SYSTEM OPCUAClient
  (* Version 1.0, Author, Eclipse 4diac *)
  APPLICATION OPCUAClientApp
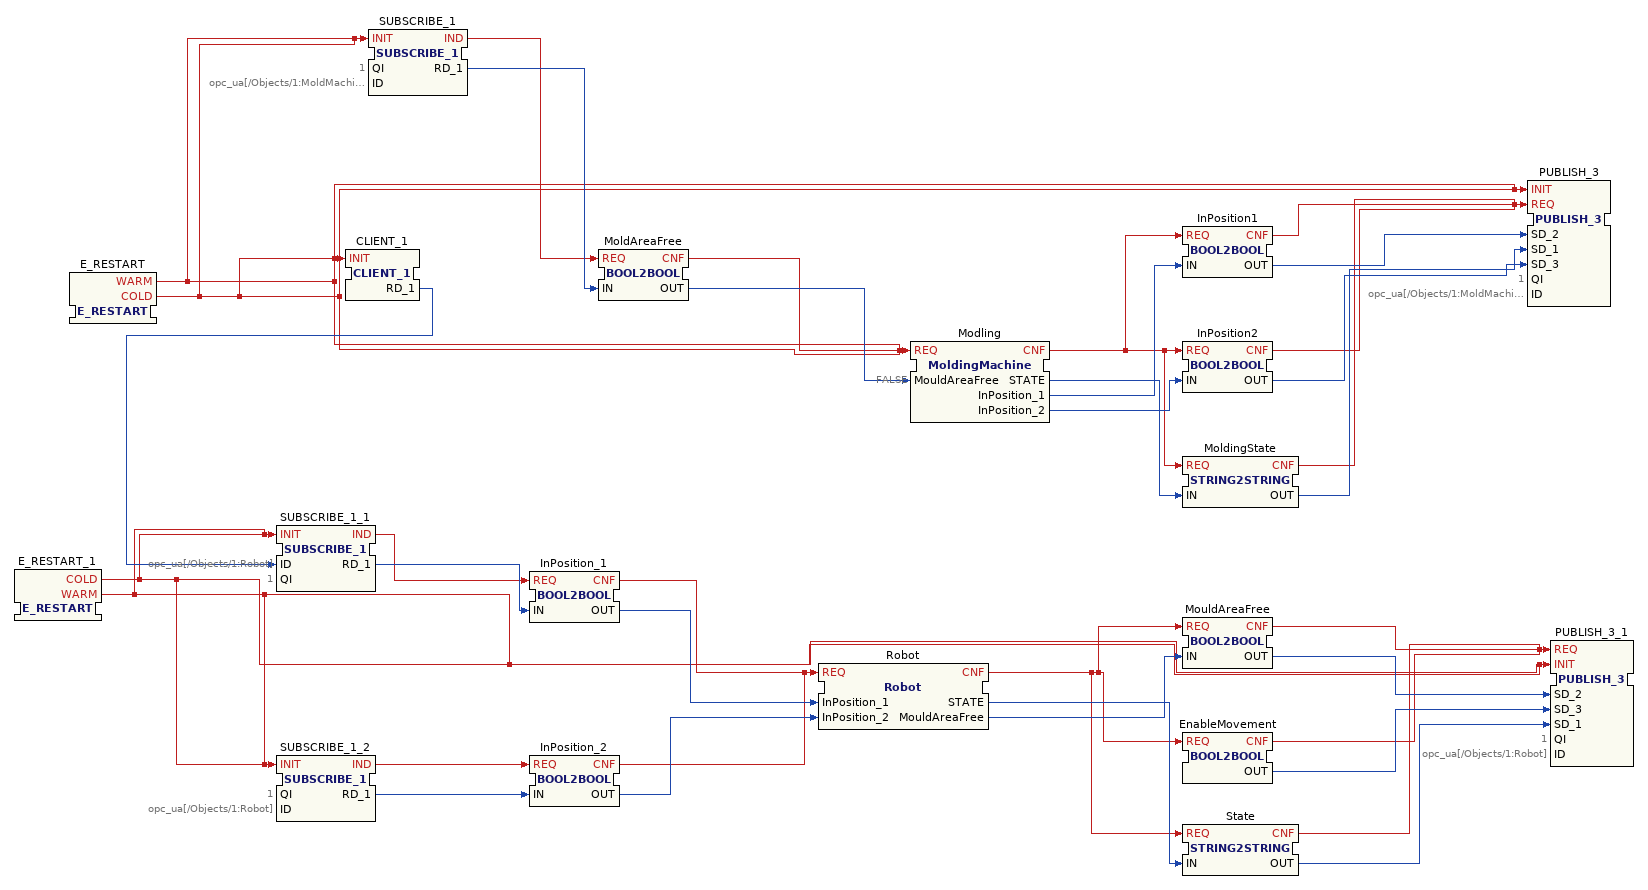
    FBS
      MoldAreaFree : BOOL2BOOL;
      E_RESTART : E_RESTART;
      SUBSCRIBE_1 : SUBSCRIBE_1(QI := 1, ID := opc_ua[/Objects/1:MoldMachine]);
      SUBSCRIBE_1_1 : SUBSCRIBE_1(QI := 1, ID := opc_ua[/Objects/1:Robot]);
      PUBLISH_3 : PUBLISH_3(QI := 1, ID := opc_ua[/Objects/1:MoldMachine]);
      Modling : MoldingMachine(MouldAreaFree := FALSE);
      InPosition_1 : BOOL2BOOL;
      SUBSCRIBE_1_2 : SUBSCRIBE_1(QI := 1, ID := opc_ua[/Objects/1:Robot]);
      InPosition_2 : BOOL2BOOL;
      PUBLISH_3_1 : PUBLISH_3(QI := 1, ID := opc_ua[/Objects/1:Robot]);
      InPosition1 : BOOL2BOOL;
      InPosition2 : BOOL2BOOL;
      MoldingState : STRING2STRING;
      MouldAreaFree : BOOL2BOOL;
      EnableMovement : BOOL2BOOL;
      State : STRING2STRING;
      Robot : Robot;
      E_RESTART_1 : E_RESTART;
      CLIENT_1 : CLIENT_1;
    END_FBS
    EVENT_CONNECTIONS
      E_RESTART.WARM TO SUBSCRIBE_1.INIT;
      E_RESTART.COLD TO SUBSCRIBE_1.INIT;
      SUBSCRIBE_1.IND TO MoldAreaFree.REQ;
      E_RESTART.COLD TO PUBLISH_3.INIT;
      E_RESTART.WARM TO PUBLISH_3.INIT;
      MoldAreaFree.CNF TO Modling.REQ;
      E_RESTART.COLD TO Modling.REQ;
      E_RESTART.WARM TO Modling.REQ;
      SUBSCRIBE_1_1.IND TO InPosition_1.REQ;
      SUBSCRIBE_1_2.IND TO InPosition_2.REQ;
      Modling.CNF TO InPosition1.REQ;
      Modling.CNF TO InPosition2.REQ;
      Modling.CNF TO MoldingState.REQ;
      InPosition1.CNF TO PUBLISH_3.REQ;
      InPosition2.CNF TO PUBLISH_3.REQ;
      MoldingState.CNF TO PUBLISH_3.REQ;
      InPosition_1.CNF TO Robot.REQ;
      InPosition_2.CNF TO Robot.REQ;
      Robot.CNF TO MouldAreaFree.REQ;
      Robot.CNF TO EnableMovement.REQ;
      Robot.CNF TO State.REQ;
      MouldAreaFree.CNF TO PUBLISH_3_1.REQ;
      EnableMovement.CNF TO PUBLISH_3_1.REQ;
      State.CNF TO PUBLISH_3_1.REQ;
      E_RESTART_1.COLD TO SUBSCRIBE_1_1.INIT;
      E_RESTART_1.COLD TO SUBSCRIBE_1_2.INIT;
      E_RESTART_1.COLD TO PUBLISH_3_1.INIT;
      E_RESTART_1.WARM TO SUBSCRIBE_1_1.INIT;
      E_RESTART_1.WARM TO SUBSCRIBE_1_2.INIT;
      E_RESTART_1.WARM TO PUBLISH_3_1.INIT;
      E_RESTART.COLD TO CLIENT_1.INIT;
      E_RESTART.WARM TO CLIENT_1.INIT;
    END_CONNECTIONS
    DATA_CONNECTIONS
      SUBSCRIBE_1.RD_1 TO MoldAreaFree.IN;
      SUBSCRIBE_1_1.RD_1 TO InPosition_1.IN;
      MoldAreaFree.OUT TO Modling.MouldAreaFree;
      SUBSCRIBE_1_2.RD_1 TO InPosition_2.IN;
      Modling.STATE TO MoldingState.IN;
      Modling.InPosition_1 TO InPosition1.IN;
      Modling.InPosition_2 TO InPosition2.IN;
      InPosition1.OUT TO PUBLISH_3.SD_2;
      MoldingState.OUT TO PUBLISH_3.SD_1;
      InPosition2.OUT TO PUBLISH_3.SD_3;
      InPosition_1.OUT TO Robot.InPosition_1;
      InPosition_2.OUT TO Robot.InPosition_2;
      Robot.STATE TO State.IN;
      Robot.MouldAreaFree TO MouldAreaFree.IN;
      MouldAreaFree.OUT TO PUBLISH_3_1.SD_2;
      EnableMovement.OUT TO PUBLISH_3_1.SD_3;
      State.OUT TO PUBLISH_3_1.SD_1;
      CLIENT_1.RD_1 TO SUBSCRIBE_1_1.ID;
    END_CONNECTIONS
  END_APPLICATION
  DEVICE Moulding : FORTE_PC(MGR_ID := "localhost:61499")
    {SET_ATTRIBUTE(Profile, HOLOBLOC)} (* device profile *)
    RESOURCE EMB_RES : EMB_RES
      FBS
        E_RESTART : E_RESTART;
        SUBSCRIBE_1 : SUBSCRIBE_1(QI := 1, ID := opc_ua[/Objects/1:MoldMachine]);
        MoldAreaFree : BOOL2BOOL;
        PUBLISH_3 : PUBLISH_3(QI := 1, ID := opc_ua[/Objects/1:MoldMachine]);
        Modling : MoldingMachine(MouldAreaFree := FALSE);
        InPosition1 : BOOL2BOOL;
        InPosition2 : BOOL2BOOL;
        MoldingState : STRING2STRING;
      END_FBS
      EVENT_CONNECTIONS
        E_RESTART.WARM TO SUBSCRIBE_1.INIT;
        E_RESTART.COLD TO SUBSCRIBE_1.INIT;
        SUBSCRIBE_1.IND TO MoldAreaFree.REQ;
        E_RESTART.COLD TO PUBLISH_3.INIT;
        E_RESTART.WARM TO PUBLISH_3.INIT;
        MoldAreaFree.CNF TO Modling.REQ;
        E_RESTART.COLD TO Modling.REQ;
        E_RESTART.WARM TO Modling.REQ;
        Modling.CNF TO InPosition1.REQ;
        InPosition1.CNF TO PUBLISH_3.REQ;
        Modling.CNF TO InPosition2.REQ;
        InPosition2.CNF TO PUBLISH_3.REQ;
        Modling.CNF TO MoldingState.REQ;
        MoldingState.CNF TO PUBLISH_3.REQ;
      END_CONNECTIONS
      DATA_CONNECTIONS
        SUBSCRIBE_1.RD_1 TO MoldAreaFree.IN;
        MoldAreaFree.OUT TO Modling.MouldAreaFree;
        Modling.InPosition_1 TO InPosition1.IN;
        InPosition1.OUT TO PUBLISH_3.SD_2;
        Modling.InPosition_2 TO InPosition2.IN;
        InPosition2.OUT TO PUBLISH_3.SD_3;
        Modling.STATE TO MoldingState.IN;
        MoldingState.OUT TO PUBLISH_3.SD_1;
      END_CONNECTIONS
    END_RESOURCE
  END_DEVICE
  DEVICE Rbobt : FORTE_PC(MGR_ID := "localhost:61500")
    {SET_ATTRIBUTE(Profile, HOLOBLOC)} (* device profile *)
    RESOURCE EMB_RES : EMB_RES
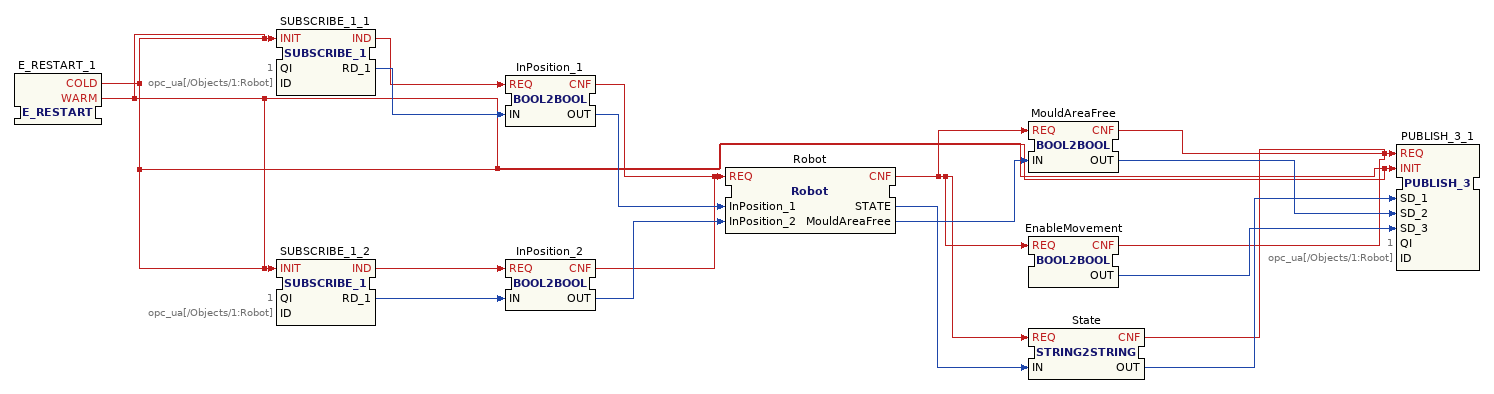
      FBS
        SUBSCRIBE_1_1 : SUBSCRIBE_1(QI := 1, ID := opc_ua[/Objects/1:Robot]);
        InPosition_1 : BOOL2BOOL;
        SUBSCRIBE_1_2 : SUBSCRIBE_1(QI := 1, ID := opc_ua[/Objects/1:Robot]);
        InPosition_2 : BOOL2BOOL;
        MouldAreaFree : BOOL2BOOL;
        State : STRING2STRING;
        EnableMovement : BOOL2BOOL;
        Robot : Robot;
        PUBLISH_3_1 : PUBLISH_3(QI := 1, ID := opc_ua[/Objects/1:Robot]);
        E_RESTART_1 : E_RESTART;
      END_FBS
      EVENT_CONNECTIONS
        SUBSCRIBE_1_1.IND TO InPosition_1.REQ;
        SUBSCRIBE_1_2.IND TO InPosition_2.REQ;
        InPosition_1.CNF TO Robot.REQ;
        InPosition_2.CNF TO Robot.REQ;
        Robot.CNF TO MouldAreaFree.REQ;
        Robot.CNF TO EnableMovement.REQ;
        Robot.CNF TO State.REQ;
        MouldAreaFree.CNF TO PUBLISH_3_1.REQ;
        EnableMovement.CNF TO PUBLISH_3_1.REQ;
        State.CNF TO PUBLISH_3_1.REQ;
        E_RESTART_1.COLD TO SUBSCRIBE_1_1.INIT;
        E_RESTART_1.COLD TO SUBSCRIBE_1_2.INIT;
        E_RESTART_1.COLD TO PUBLISH_3_1.INIT;
        E_RESTART_1.WARM TO SUBSCRIBE_1_1.INIT;
        E_RESTART_1.WARM TO SUBSCRIBE_1_2.INIT;
        E_RESTART_1.WARM TO PUBLISH_3_1.INIT;
      END_CONNECTIONS
      DATA_CONNECTIONS
        SUBSCRIBE_1_1.RD_1 TO InPosition_1.IN;
        SUBSCRIBE_1_2.RD_1 TO InPosition_2.IN;
        InPosition_1.OUT TO Robot.InPosition_1;
        InPosition_2.OUT TO Robot.InPosition_2;
        Robot.STATE TO State.IN;
        Robot.MouldAreaFree TO MouldAreaFree.IN;
        State.OUT TO PUBLISH_3_1.SD_1;
        MouldAreaFree.OUT TO PUBLISH_3_1.SD_2;
        EnableMovement.OUT TO PUBLISH_3_1.SD_3;
      END_CONNECTIONS
    END_RESOURCE
  END_DEVICE
  MAPPINGS
    OPCUAClientApp.E_RESTART ON Moulding.EMB_RES.E_RESTART;
    OPCUAClientApp.SUBSCRIBE_1 ON Moulding.EMB_RES.SUBSCRIBE_1;
    OPCUAClientApp.MoldAreaFree ON Moulding.EMB_RES.MoldAreaFree;
    OPCUAClientApp.PUBLISH_3 ON Moulding.EMB_RES.PUBLISH_3;
    OPCUAClientApp.Modling ON Moulding.EMB_RES.Modling;
    OPCUAClientApp.InPosition1 ON Moulding.EMB_RES.InPosition1;
    OPCUAClientApp.InPosition2 ON Moulding.EMB_RES.InPosition2;
    OPCUAClientApp.MoldingState ON Moulding.EMB_RES.MoldingState;
    OPCUAClientApp.SUBSCRIBE_1_1 ON Rbobt.EMB_RES.SUBSCRIBE_1_1;
    OPCUAClientApp.InPosition_1 ON Rbobt.EMB_RES.InPosition_1;
    OPCUAClientApp.SUBSCRIBE_1_2 ON Rbobt.EMB_RES.SUBSCRIBE_1_2;
    OPCUAClientApp.InPosition_2 ON Rbobt.EMB_RES.InPosition_2;
    OPCUAClientApp.MouldAreaFree ON Rbobt.EMB_RES.MouldAreaFree;
    OPCUAClientApp.State ON Rbobt.EMB_RES.State;
    OPCUAClientApp.EnableMovement ON Rbobt.EMB_RES.EnableMovement;
    OPCUAClientApp.Robot ON Rbobt.EMB_RES.Robot;
    OPCUAClientApp.PUBLISH_3_1 ON Rbobt.EMB_RES.PUBLISH_3_1;
    OPCUAClientApp.E_RESTART_1 ON Rbobt.EMB_RES.E_RESTART_1;
  END_MAPPINGS
  SEGMENTS
    Ethernet : Ethernet;
  END_SEGMENTS
  LINKS
    Moulding => Ethernet;
    Rbobt => Ethernet;
  END_LINKS
END_SYSTEM
